// TwinCAT 3 PLC project Sample02
// ProgramVersion: 3.1.4020.10
// libraries:
//   Tc2_Standard, * (Beckhoff Automation GmbH)
//   Tc2_System, * (Beckhoff Automation GmbH)
//   Tc3_Module, * (Beckhoff Automation GmbH)
// project tree:
//   / PlcTask.TcTTO (not stored)
//   POUs/ Class Diagram.TcCD (not stored), FB_AnalogValue.TcPOU (not stored), FB_Controller.TcPOU, FB_Lamp.TcPOU (not stored), FB_LampSetDirectDALI.TcPOU, FB_LampOnOffAdapter.TcPOU (not stored), FB_LampSetDirectAdapter.TcPOU (not stored), FB_LampSetDirectDALIAdapter.TcPOU, FB_LampUpDown.TcPOU (not stored), FB_LampSetDirect.TcPOU (not stored), FB_LampOnOff.TcPOU (not stored), FB_LampUpDownAdapter.TcPOU (not stored), I_OperatingTime.TcIO, I_Lamp.TcIO (not stored), I_Observer.TcIO (not stored), I_Subject.TcIO (not stored), MAIN.TcPOU (not stored)
// real-time tasks:
//   TASK PlcTask: cycle T#10ms, priority 20, ADS port 350

// ---- POUs/I_OperatingTime.TcIO
INTERFACE I_OperatingTime EXTENDS __SYSTEM.IQueryInterface

PROPERTY nOperatingTime : DINT // Operating Time [s]
GET
END_GET
SET
END_SET
END_PROPERTY

END_INTERFACE

// ---- POUs/FB_Controller.TcPOU
FUNCTION_BLOCK PUBLIC FB_Controller
VAR
	fbActualValue		: FB_AnalogValue;
	_refActiveLamp		: REFERENCE TO FB_Lamp;
END_VAR

IF (__ISVALIDREF(_refActiveLamp)) THEN
	_refActiveLamp();
END_IF

// Reduces the control value by 5 in the range of 10 to 100.
METHOD PUBLIC DimDown
IF (__ISVALIDREF(_refActiveLamp)) THEN
	_refActiveLamp.DimDown();
END_IF
END_METHOD

// Increments the control value by 5 in the range of 10 to 100.
METHOD PUBLIC DimUp
IF (__ISVALIDREF(_refActiveLamp)) THEN
	_refActiveLamp.DimUp();
END_IF
END_METHOD

{attribute 'monitoring' := 'call'}
PROPERTY PUBLIC nOperatingTime : DINT
GET
VAR
	ipOperatingTime 			: I_OperatingTime;
END_VAR
IF (__ISVALIDREF(_refActiveLamp)) THEN	
	IF (__QUERYINTERFACE(_refActiveLamp, ipOperatingTime)) THEN
		nOperatingTime := ipOperatingTime.nOperatingTime;
	ELSE
		nOperatingTime := -1; // service not supported
	END_IF
END_IF
END_GET
SET
VAR
	ipOperatingTime 			: I_OperatingTime;
END_VAR
IF (__ISVALIDREF(_refActiveLamp)) THEN	
	IF (__QUERYINTERFACE(_refActiveLamp, ipOperatingTime)) THEN
		ipOperatingTime.nOperatingTime := nOperatingTime;
	END_IF
END_IF
END_SET
END_PROPERTY

// Sets the control value to 0.
METHOD PUBLIC Off
IF (__ISVALIDREF(_refActiveLamp)) THEN
	_refActiveLamp.Off();
END_IF
END_METHOD

// Sets the control value to 100.
METHOD PUBLIC On
IF (__ISVALIDREF(_refActiveLamp)) THEN
	_refActiveLamp.On();
END_IF
END_METHOD

{attribute 'monitoring' := 'call'}
PROPERTY PUBLIC refActiveLamp : REFERENCE TO FB_Lamp
GET
refActiveLamp REF= _refActiveLamp;
END_GET
SET
IF (__ISVALIDREF(_refActiveLamp)) THEN
	_refActiveLamp.Detach();
END_IF

_refActiveLamp REF= refActiveLamp;

IF (__ISVALIDREF(refActiveLamp)) THEN
	refActiveLamp.Attach(fbActualValue);
END_IF
END_SET
END_PROPERTY

END_FUNCTION_BLOCK

// ---- POUs/FB_LampSetDirectDALI.TcPOU
FUNCTION_BLOCK PUBLIC FB_LampSetDirectDALI
VAR
	nLightLevel			: BYTE;
	_nOperatingTime		: DINT;
	tonDelay			: TON;
END_VAR

IF (nLightLevel > 0) THEN
	tonDelay(IN := TRUE, PT := T#1S);
	IF (tonDelay.Q) THEN
		tonDelay(IN := FALSE);
		_nOperatingTime := _nOperatingTime + 1;
	END_IF
ELSE
	tonDelay(IN := FALSE);
END_IF

{attribute 'monitoring' := 'call'}
PROPERTY PUBLIC nOperatingTime : DINT
GET
nOperatingTime := _nOperatingTime;
END_GET
SET
_nOperatingTime := nOperatingTime;
END_SET
END_PROPERTY

// Sets the control value of the DALI lamp to a value between 0 and 254.
METHOD PUBLIC SetLightLevel
VAR_INPUT
	nNewLightLevel		: BYTE(0..254);
END_VAR
nLightLevel := nNewLightLevel;
END_METHOD

END_FUNCTION_BLOCK

// ---- POUs/FB_LampSetDirectDALIAdapter.TcPOU
FUNCTION_BLOCK PUBLIC FB_LampSetDirectDALIAdapter EXTENDS FB_Lamp IMPLEMENTS I_OperatingTime
VAR
	fbLampSetDirectDALI		: FB_LampSetDirectDALI;
END_VAR

fbLampSetDirectDALI();

// Reduces the control value by 5 in the range of 10 to 254.
METHOD PUBLIC DimDown
IF (fbLampSetDirectDALI.nLightLevel >= 38.1) THEN
	fbLampSetDirectDALI.SetLightLevel(TO_BYTE(fbLampSetDirectDALI.nLightLevel - 12.7));
END_IF
IF (_ipObserver <> 0) THEN
	_ipObserver.Update(TO_BYTE(fbLampSetDirectDALI.nLightLevel * 100.0 / 254.0));
END_IF
END_METHOD

// Increments the control value by 5 in the range of 10 to 254.
METHOD PUBLIC DimUp
IF (fbLampSetDirectDALI.nLightLevel <= 241.3) THEN
	fbLampSetDirectDALI.SetLightLevel(TO_BYTE(TO_LREAL(fbLampSetDirectDALI.nLightLevel) + 12.7));
END_IF
IF (_ipObserver <> 0) THEN
	_ipObserver.Update(TO_BYTE(fbLampSetDirectDALI.nLightLevel * 100.0 / 254.0));
END_IF
END_METHOD

{attribute 'monitoring' := 'call'}
PROPERTY PUBLIC nOperatingTime : DINT
GET
nOperatingTime := fbLampSetDirectDALI.nOperatingTime;
END_GET
SET
fbLampSetDirectDALI.nOperatingTime := nOperatingTime;
END_SET
END_PROPERTY

// Sets the control value to 0.
METHOD PUBLIC Off
fbLampSetDirectDALI.SetLightLevel(0);
IF (_ipObserver <> 0) THEN
	_ipObserver.Update(TO_BYTE(fbLampSetDirectDALI.nLightLevel * 100.0 / 254.0));
END_IF
END_METHOD

// Sets the control value to 254.
METHOD PUBLIC On
fbLampSetDirectDALI.SetLightLevel(254);
IF (_ipObserver <> 0) THEN
	_ipObserver.Update(TO_BYTE(fbLampSetDirectDALI.nLightLevel * 100.0 / 254.0));
END_IF
END_METHOD

END_FUNCTION_BLOCK
